FUNCTION_BLOCK FB_Chamber1SpinAxisJogCWServices EXTENDS FB_ServiceBase
VAR_INPUT
	Param : ST_Chamber1SpinAxisJogParam;
	Axis_BaseUnit : I_Axis_BaseUnit;
END_VAR

M_UpdateService(CompletionBehavior := E_ServiceCompletionBehavior.ExecuteUntilExternalStop);

METHOD PROTECTED H_OnAborted
VAR_INPUT
	bFirstScan	: BOOL;
END_VAR
// Release defensively in case an unexpected transition skipped cleanup.
Axis_BaseUnit.M_ReleaseResource(OwnerId := ServiceId);
END_METHOD

METHOD PROTECTED H_OnAborting : E_PackMLHookResult
VAR_INPUT
	bFirstScan	: BOOL;
END_VAR
H_OnAborting := E_PackMLHookResult.Done;

// A Service that never acquired the Resource must not affect its Owner.
IF NOT Axis_BaseUnit.M_IsResourceOwner(OwnerId := ServiceId) THEN
	RETURN;
END_IF

Axis_BaseUnit.M_Jog(
	OwnerId:= ServiceId,
	JogForward:= FALSE, 
	JogBackwards:= FALSE, 
	Mode:= E_JogMode.MC_JOGMODE_CONTINOUS,
	Position:= Param.Position,
	Velocity:= Param.Velocity,
	Acceleration:= Param.Acceleration,
	Deceleration:= Param.Deceleration);

// Jog has no asynchronous abort phase once both direction commands are false.
Axis_BaseUnit.M_ReleaseResource(OwnerId := ServiceId);
END_METHOD

METHOD PROTECTED H_OnClearing : E_PackMLHookResult
VAR_INPUT
	bFirstScan	: BOOL;
END_VAR

VAR
	bServoOn : BOOL;
	bError : BOOL;
	nErrorId : UDINT;
END_VAR
M_ClearAllError();
H_OnClearing := E_PackMLHookResult.Done;
END_METHOD

METHOD PROTECTED H_OnComplete
VAR_INPUT
	bFirstScan	: BOOL;
END_VAR
// Completing normally releases first; this is an idempotent safety net.
Axis_BaseUnit.M_ReleaseResource(OwnerId := ServiceId);
END_METHOD

METHOD PROTECTED H_OnCompleting : E_PackMLHookResult
VAR_INPUT
	bFirstScan	: BOOL;
END_VAR
Axis_BaseUnit.M_Jog(
	OwnerId:= ServiceId,
	JogForward:= FALSE, 
	JogBackwards:= FALSE, 
	Mode:= E_JogMode.MC_JOGMODE_CONTINOUS,
	Position:= Param.Position,
	Velocity:= Param.Velocity,
	Acceleration:= Param.Acceleration,
	Deceleration:= Param.Deceleration);

// Release only after the active Jog request has been withdrawn.
Axis_BaseUnit.M_ReleaseResource(OwnerId := ServiceId);
H_OnCompleting := E_PackMLHookResult.Done;
END_METHOD

METHOD PROTECTED H_OnExecute : E_PackMLHookResult
VAR_INPUT
	bFirstScan	: BOOL;
END_VAR

VAR
	bError : BOOL;
	nErrorId : UDINT;
END_VAR
H_OnExecute := E_PackMLHookResult.Busy;

Axis_BaseUnit.M_Jog(
	OwnerId:= ServiceId,
	JogForward:= TRUE,
	JogBackwards:= FALSE,
	Mode:= E_JogMode.MC_JOGMODE_CONTINOUS,
	Position:= Param.Position,
	Velocity:= Param.Velocity,
	Acceleration:= Param.Acceleration,
	Deceleration:= Param.Deceleration,
	Done=> , Error=> bError, ErrorId=> nErrorId);


IF bError THEN
	M_AddError(
		MainErrorId := E_Chamber1ErrorCode.Axis_Command_Error_During_Execute,
		SourceErrorId := nErrorId,
		Message := 'Jog failed during Execute.');
	RequestCommand(E_PackMLCommand.Abort);
END_IF
END_METHOD

METHOD PROTECTED H_OnIdle
VAR_INPUT
	bFirstScan	: BOOL;
END_VAR
// Idle Services must not retain a Resource from an earlier operation.
Axis_BaseUnit.M_ReleaseResource(OwnerId := ServiceId);
END_METHOD

METHOD PROTECTED H_OnResetting : E_PackMLHookResult
VAR_INPUT
	bFirstScan	: BOOL;
END_VAR
H_OnResetting := E_PackMLHookResult.Done;
END_METHOD

METHOD PROTECTED H_OnStarting : E_PackMLHookResult
VAR_INPUT
	bFirstScan	: BOOL;
END_VAR
H_OnStarting := E_PackMLHookResult.Busy;

// Validate Service-owned data before reserving the shared BaseUnit.
IF Param.Velocity <= 0 THEN
	M_AddError(MainErrorId := E_Chamber1ErrorCode.Invalid_Param, SourceErrorId := 0, Message := 'Velocity must be greater than zero.');
	RequestCommand(E_PackMLCommand.Abort);
	RETURN;
END_IF

IF Param.Acceleration < 0 THEN
	M_AddError(MainErrorId := E_Chamber1ErrorCode.Invalid_Param, SourceErrorId := 0, Message := 'Acceleration must not be negative.');
	RequestCommand(E_PackMLCommand.Abort);
	RETURN;
END_IF

IF Param.Deceleration < 0 THEN
	M_AddError(MainErrorId := E_Chamber1ErrorCode.Invalid_Param, SourceErrorId := 0, Message := 'Deceleration must not be negative.');
	RequestCommand(E_PackMLCommand.Abort);
	RETURN;
END_IF

// Resource contention is a failed Start, not a wait condition.
IF NOT Axis_BaseUnit.M_AcquireResource(OwnerId := ServiceId) THEN
	M_AddError(MainErrorId := E_Chamber1ErrorCode.Resource_Acquire_Failed_During_Starting, SourceErrorId := 0, Message := 'Axis resource acquisition failed during Starting.');
	RequestCommand(E_PackMLCommand.Abort);
	RETURN;
END_IF

// Physical checks occur only after this Service owns the BaseUnit.
IF Axis_BaseUnit.AxisIsDisabled THEN
	M_AddError(MainErrorId := E_Chamber1ErrorCode.Axis_Not_Servo_On_During_Starting, SourceErrorId := 0, Message := 'Axis is not servo on during Starting.');
	RequestCommand(E_PackMLCommand.Abort);
	RETURN;
END_IF

IF Axis_BaseUnit.AxisHasJob THEN
	M_AddError(MainErrorId := E_Chamber1ErrorCode.Axis_Is_Busy_During_Starting, SourceErrorId := 0, Message := 'Axis is busy during Starting.');
	RequestCommand(E_PackMLCommand.Abort);
	RETURN;
END_IF

H_OnStarting := E_PackMLHookResult.Done;
END_METHOD

METHOD PROTECTED H_OnStopped
VAR_INPUT
	bFirstScan	: BOOL;
END_VAR
// Release defensively after every Stop path.
Axis_BaseUnit.M_ReleaseResource(OwnerId := ServiceId);
END_METHOD

METHOD PROTECTED H_OnStopping : E_PackMLHookResult
VAR_INPUT
	bFirstScan	: BOOL;
END_VAR
H_OnStopping := E_PackMLHookResult.Done;

// Resource acquisition failures enter Stopping without owning the Axis.
IF NOT Axis_BaseUnit.M_IsResourceOwner(OwnerId := ServiceId) THEN
	RETURN;
END_IF

Axis_BaseUnit.M_Jog(
	OwnerId:= ServiceId,
	JogForward:= FALSE, 
	JogBackwards:= FALSE, 
	Mode:= E_JogMode.MC_JOGMODE_CONTINOUS,
	Position:= Param.Position,
	Velocity:= Param.Velocity,
	Acceleration:= Param.Acceleration,
	Deceleration:= Param.Deceleration);

// Jog is stopped once both direction commands have been withdrawn.
Axis_BaseUnit.M_ReleaseResource(OwnerId := ServiceId);
END_METHOD

END_FUNCTION_BLOCK

(* stored: Version 1.1.0.1, ProductVersion 3.1.4026.18
   POU FB_Chamber1SpinAxisJogCWServices: Id {a61ac5cd-09b6-4f2d-bc54-d014db7401a2}, SpecialFunc None
   Folder StateAction: Id {30486db3-fa54-4a70-b426-5f8ba9d0504f}
   Method H_OnAborted: Id {b48428e2-059a-4878-a27b-576d41f2ba26}
   Method H_OnAborting: Id {df4c7f2d-8a88-4d35-a321-0716e918b536}
   Method H_OnClearing: Id {9a60118e-19f9-4bca-893b-e890bf0b19c9}
   Method H_OnComplete: Id {fd680a59-d09e-4091-ac1f-b02ebd6a48e6}
   Method H_OnCompleting: Id {61491643-adf6-4106-831a-f4dfe9e14738}
   Method H_OnExecute: Id {2dba6e2e-7918-46c6-a0b6-50da9e5cf338}
   Method H_OnIdle: Id {801e1204-bf1d-4d12-b7fd-e2791384226a}
   Method H_OnResetting: Id {cd0cb289-d0f8-442c-af15-52d2005bf619}
   Method H_OnStarting: Id {bcd7c333-82d2-481d-9c52-d49b2030a18e}
   Method H_OnStopped: Id {7643e72d-21d0-42a9-a466-1828d294ec10}
   Method H_OnStopping: Id {7e40e9e4-ecf0-49b7-86b3-13897394333e} *)
